(*			
	RafalOS
	Rafał Osajda		20.11.2025		TC 4024.66
	Moduł przygotowania danych dla Okna głównego w trybie konserwacji
*)
FUNCTION_BLOCK FB_MCHMIPrepareDataForScreen_00_02 EXTENDS FB_MCHMIPrepareDataForScreen IMPLEMENTS ITF_MCHMIPrepareDataForScreen
VAR
END_VAR

(*			
	RafalOS
	Rafał Osajda		19.11.2025		TC 4024.66
	Czyści danych przy zmienia ramki po poprzedniej ramce
*)
METHOD PUBLIC ClearAfterScreen : BOOL
VAR_INPUT
END_VAR
SUPER^.ClearAfterScreen ();
END_METHOD

(*			
	RafalOS
	Rafał Osajda		14.11.2025		TC 4024.66
	Metoda przygotowywania danych dla HMI 
	W niej odbywa się odpytywanie właściego elementu przez łącznik
*)
METHOD PUBLIC PrepareDataForHMI : BOOL
VAR_INPUT
END_VAR
SUPER^.PrepareDataForHMI ();
END_METHOD

(*			
	RafalOS
	Rafał Osajda		19.11.2025		TC 4024.66
	Przygotowanie ramki pood tamke do wyświetlenia - tylko przygotowanie a nie przygotowanie danych do wyświetlenia
*)
METHOD PUBLIC PrepareForScreen : BOOL
VAR_INPUT
END_VAR
SUPER^.PrepareForScreen ();
END_METHOD

END_FUNCTION_BLOCK

(* stored: Version 1.1.0.1
   POU FB_MCHMIPrepareDataForScreen_00_02: Id {c2e13f1c-fddd-0c70-1b16-9d11e2f022e9}, SpecialFunc None
   Folder ITF_PDFS: Id {9b0edb78-a6a2-0099-03bd-9a3d5c88d819}
   Method ClearAfterScreen: Id {e2eb0b74-915e-03bd-39a3-3839ad5f96b4}
   Method PrepareDataForHMI: Id {0be6b2c1-4996-018a-33cd-9018bbc82f0e}
   Method PrepareForScreen: Id {edde4ebf-8061-05b0-31d0-b3835fc938fb} *)
